TYPE E_MotorDirection :
(
	NoDirection := 0,
	OnlyPostive,
	OnlyNegative,
	Two_Way
)INT;
END_TYPE

(* stored: Version 1.1.0.1, ProductVersion 3.1.4024.11
   DUT E_MotorDirection: Id {f22319e8-7b97-41bb-bdb3-3ddc86c6387e} *)
